TYPE ST_DamperMotionConfig :
STRUCT
    stX : ST_VelocityConfig;
    stY : ST_VelocityConfig;
    stZ : ST_VelocityConfig;
    fPositionTolerance : LREAL;
    stRotation : ST_DamperRotationMotionConfig;
    tMoveTimeout : TIME; // 单次自动运动超时，统一在GVL_MotionConfig赋值
END_STRUCT
END_TYPE

(* stored: Version 1.1.0.1, ProductVersion 3.1.4026.20
   DUT ST_DamperMotionConfig: Id {d8745e73-ef26-4ac8-bbea-7b100b470e35} *)
